{attribute addProperty BoxType "KL2300-0100"}
{attribute addProperty Id "Channel_1Channel_B8364C2500Channel_2Channel_B8364C2500Channel_3Channel_B8364C2500Channel_4Channel_B8364C2500"}
{attribute addProperty CRC "1540156748"}
{attribute addProperty SizeInBites "0"}
{attribute addProperty SizeInBytes "0"}
TYPE KL_5BCCED4C :
STRUCT
	{attribute addProperty Name "Channel_1"}
	Channel_1 : Channel_B8364C25;
	{attribute addProperty Name "Channel_2"}
	Channel_2 : Channel_B8364C25;
	{attribute addProperty Name "Channel_3"}
	Channel_3 : Channel_B8364C25;
	{attribute addProperty Name "Channel_4"}
	Channel_4 : Channel_B8364C25;
END_STRUCT
END_TYPE

(* stored: Version 1.2.0.0, ProductVersion 3.1.4024.9
   DUT KL_5BCCED4C: Id {d092b05e-e972-471b-8d9d-381bef45db33} *)
